// SIMATIC S7-200 project (STEP 7-Micro/WIN), CPU 221 REL 01.10

SYMBOL_TABLE SYM1
First_Scan_On    SM0.1    // This bit is on for the first scan cycle only.
PLS0_Ctrl        SMB67    // Controls pulse train output & pulse width modulation functions for output Q0.0.
PTO0_Profile     SMW168   // Start of profile table, pulse train output 0, expressed as byte offset from V0.
END_SYMBOL_TABLE

ORGANIZATION_BLOCK MAIN:OB1
TITLE=
BEGIN
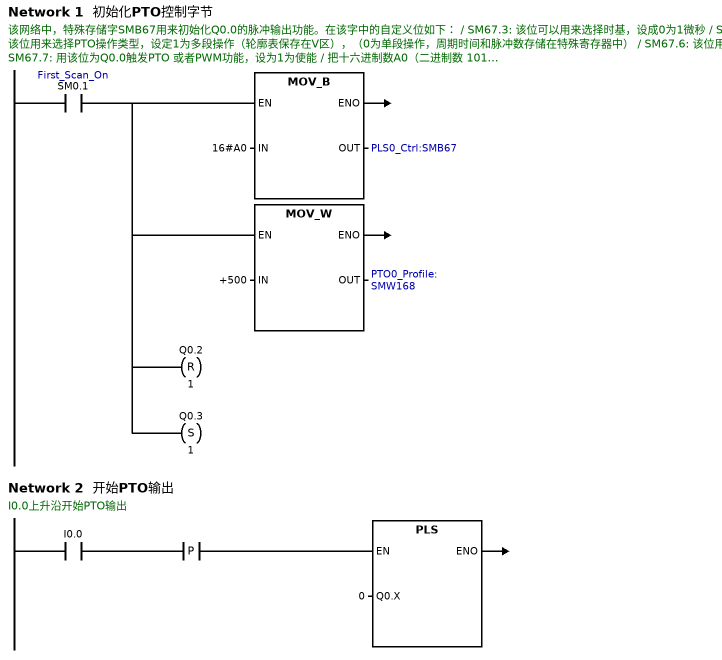
Network 1 // 初始化PTO控制字节
// 该网络中，特殊存储字SMB67用来初始化Q0.0的脉冲输出功能。在该字中的自定义位如下：
// SM67.3: 该位可以用来选择时基，设成0为1微秒
// SM67.4: 该位用来选择修正方法，设定0为异步修正（1为同步修正）
// SM67.5: 该位用来选择PTO操作类型，设定1为多段操作（轮廓表保存在V区），（0为单段操作，周期时间和脉冲数存储在特殊寄存器中）
// SM67.6: 该位用来为Q0.0选择PTO或者PWM功能，设为0选择PTO模式（1是PWM模式）
// SM67.7: 用该位为Q0.0触发PTO 或者PWM功能，设为1为使能
// 把十六进制数A0（二进制数 1010 0000）移到特殊寄存字SMB67，含义是设定时基为1微秒，选择异步修正，选择多段操作，选择PTO模式，使能在可变寄存区读取斜坡轮廓，使能输出Q0.0
// 把常数500移入特殊寄存字SMW168，在V区选择Q0.0 PTO寄存区（Q0.0 PTO斜坡轮廓表开始于VB500）
// 重新设置输出Q0.2来使能顺时针方向旋转
// 设置输出Q0.3来使能功率部分
// During the first scan cycle only,
// set up the PTO control byte
// as follows:
// Time base = 1 microsecond
// per tick.
// Select asynchronous update.
// Read ramp profile in V memory.
// Select PTO mode.
// Enable output Q0.0 for PTO
// or PWM.
// Load the pointer to
// the PTO profile 
// in V memory (Q0.0 PTO ramp
// profile table starts at VB500).
// Enable clockwise rotation.
// Enable the power section.
LD     First_Scan_On:SM0.1
MOVB   16#A0, PLS0_Ctrl:SMB67
MOVW   +500, PTO0_Profile:SMW168
R      Q0.2, 1
S      Q0.3, 1
Network 2 // 开始PTO输出
// I0.0上升沿开始PTO输出
// If there is a positive transition
// (Edge Up)
// at input bit I0.0,
// start the Q0.0 PTO ramp profile.
LD     I0.0
EU
PLS    0
END_ORGANIZATION_BLOCK

DATA_BLOCK_TAB 用户定义1
BEGIN
// 输出Q0.0PTO功能的斜坡轮廓表：
VB500    3                   // 段数为3
// 第一段    
VW501    500                 // 500ms（2kHz）循环周期开始
VW503    -2                  // 每个脉冲降低2ms
VD505    200                 // 200个脉冲
// 第二段
VW509    100                 // 100ms（10kHz）的固定循环周期
VW511    0
VD513    3400                // 3400个脉冲
// 第三段
VW517    100                 // 100ms循环周期
VW519    1                   // 每个脉冲增加1ms( 最终速度 = 2 kHz)
VD521    400                 // 400个脉冲
END_DATA_BLOCK_TAB
